// Mitsubishi GX Works2 project: 0708   PLC: Q02/Q02H

PROGRAM MAIN
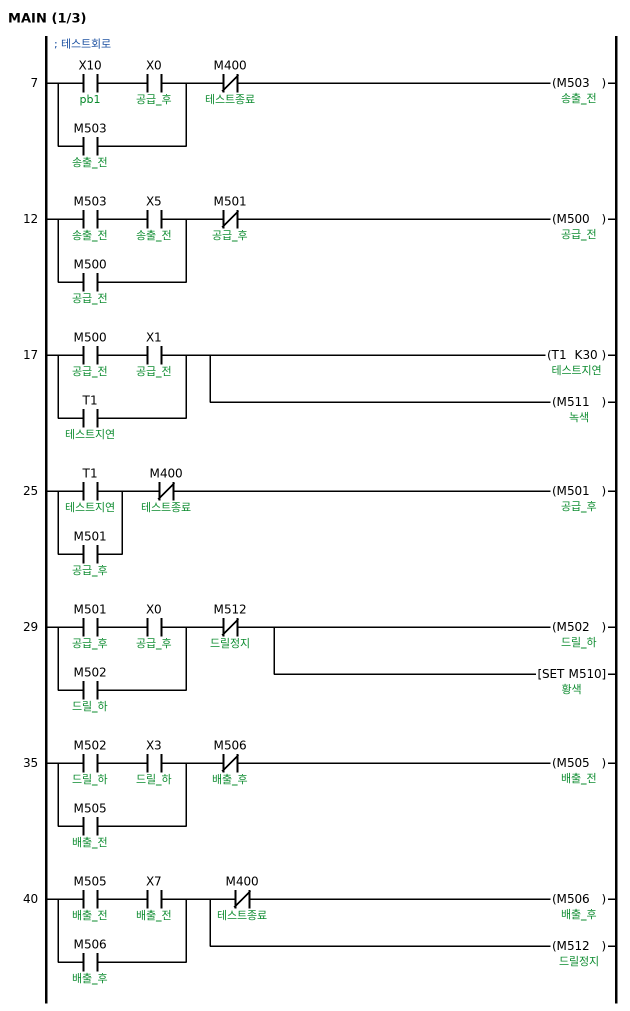
; 테스트회로
7     LD      X10  ; pb1
      AND     X0  ; 공급_후
      OR      M503  ; 송출_전
      ANI     M400  ; 테스트종료
      OUT     M503  ; 송출_전
12    LD      M503  ; 송출_전
      AND     X5  ; 송출_전
      OR      M500  ; 공급_전
      ANI     M501  ; 공급_후
      OUT     M500  ; 공급_전
17    LD      M500  ; 공급_전
      AND     X1  ; 공급_전
      OR      T1  ; 테스트지연
      OUT     T1 K30  ; 테스트지연
      OUT     M511  ; 녹색
25    LD      T1  ; 테스트지연
      OR      M501  ; 공급_후
      ANI     M400  ; 테스트종료
      OUT     M501  ; 공급_후
29    LD      M501  ; 공급_후
      AND     X0  ; 공급_후
      OR      M502  ; 드릴_하
      ANI     M512  ; 드릴정지
      OUT     M502  ; 드릴_하
      SET     M510  ; 황색
35    LD      M502  ; 드릴_하
      AND     X3  ; 드릴_하
      OR      M505  ; 배출_전
      ANI     M506  ; 배출_후
      OUT     M505  ; 배출_전
40    LD      M505  ; 배출_전
      AND     X7  ; 배출_전
      OR      M506  ; 배출_후
      MPS
      ANI     M400  ; 테스트종료
      OUT     M506  ; 배출_후
      MPP
      OUT     M512  ; 드릴정지
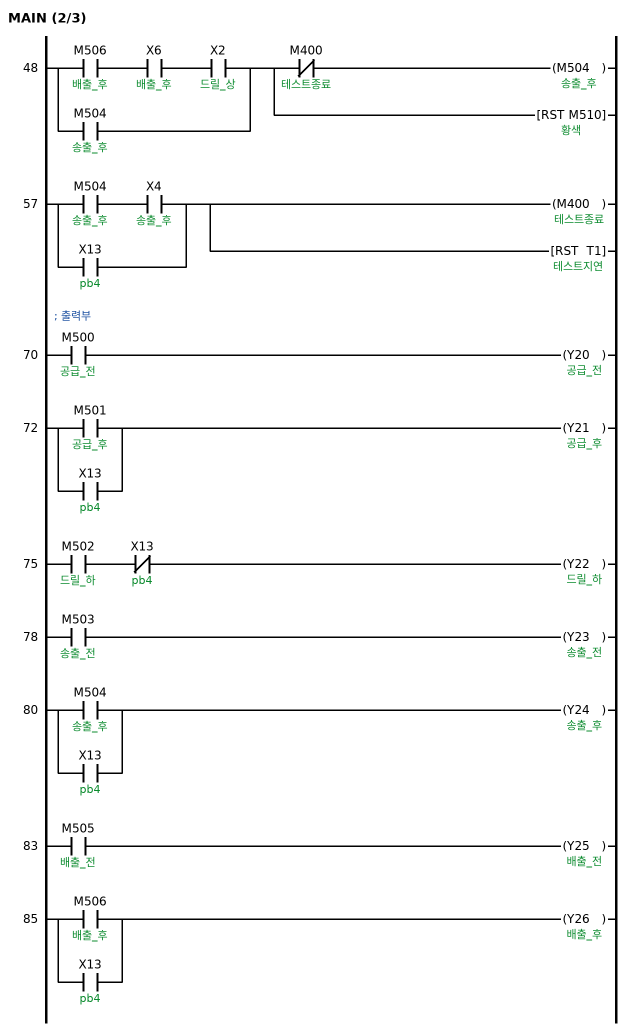
48    LD      M506  ; 배출_후
      AND     X6  ; 배출_후
      AND     X2  ; 드릴_상
      OR      M504  ; 송출_후
      MPS
      ANI     M400  ; 테스트종료
      OUT     M504  ; 송출_후
      MPP
      RST     M510  ; 황색
57    LD      M504  ; 송출_후
      AND     X4  ; 송출_후
      OR      X13  ; pb4
      OUT     M400  ; 테스트종료
      RST     T1  ; 테스트지연
; 출력부
70    LD      M500  ; 공급_전
      OUT     Y20  ; 공급_전
72    LD      M501  ; 공급_후
      OR      X13  ; pb4
      OUT     Y21  ; 공급_후
75    LD      M502  ; 드릴_하
      ANI     X13  ; pb4
      OUT     Y22  ; 드릴_하
78    LD      M503  ; 송출_전
      OUT     Y23  ; 송출_전
80    LD      M504  ; 송출_후
      OR      X13  ; pb4
      OUT     Y24  ; 송출_후
83    LD      M505  ; 배출_전
      OUT     Y25  ; 배출_전
85    LD      M506  ; 배출_후
      OR      X13  ; pb4
      OUT     Y26  ; 배출_후
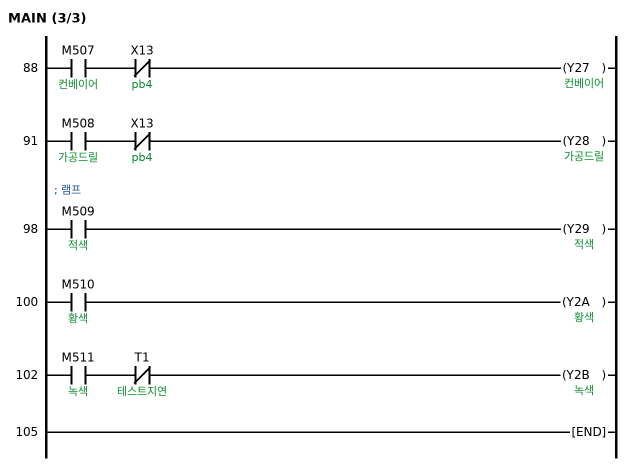
88    LD      M507  ; 컨베이어
      ANI     X13  ; pb4
      OUT     Y27  ; 컨베이어
91    LD      M508  ; 가공드릴
      ANI     X13  ; pb4
      OUT     Y28  ; 가공드릴
; 램프
98    LD      M509  ; 적색
      OUT     Y29  ; 적색
100   LD      M510  ; 황색
      OUT     Y2A  ; 황색
102   LD      M511  ; 녹색
      ANI     T1  ; 테스트지연
      OUT     Y2B  ; 녹색
105   END
END_PROGRAM

PROGRAM MAIN1
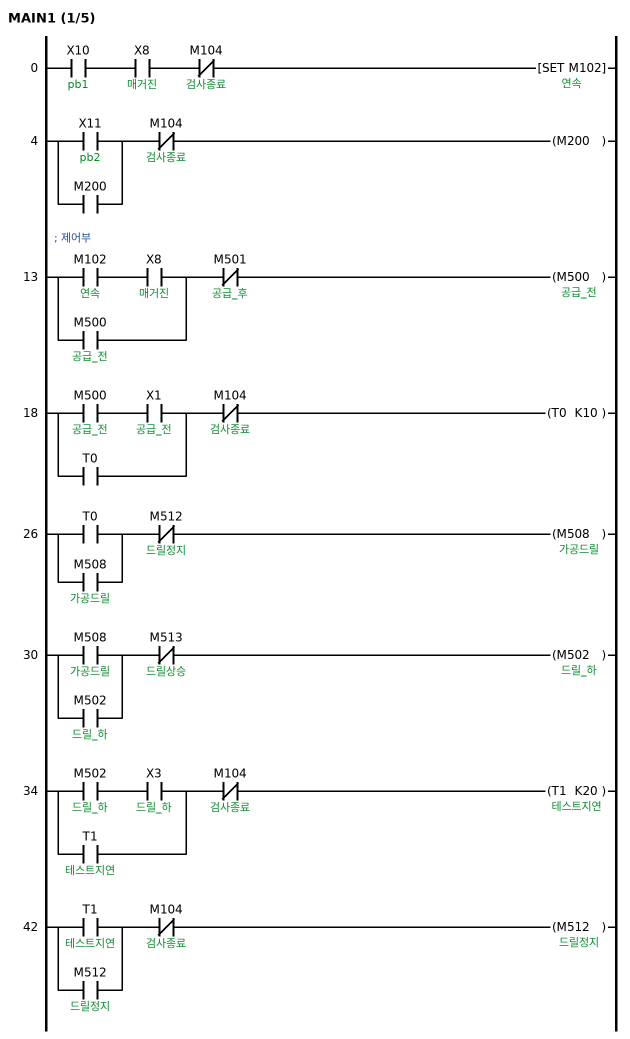
0     LD      X10  ; pb1
      AND     X8  ; 매거진
      ANI     M104  ; 검사종료
      SET     M102  ; 연속
4     LD      X11  ; pb2
      OR      M200
      ANI     M104  ; 검사종료
      OUT     M200
; 제어부
13    LD      M102  ; 연속
      AND     X8  ; 매거진
      OR      M500  ; 공급_전
      ANI     M501  ; 공급_후
      OUT     M500  ; 공급_전
18    LD      M500  ; 공급_전
      AND     X1  ; 공급_전
      OR      T0
      ANI     M104  ; 검사종료
      OUT     T0 K10
26    LD      T0
      OR      M508  ; 가공드릴
      ANI     M512  ; 드릴정지
      OUT     M508  ; 가공드릴
30    LD      M508  ; 가공드릴
      OR      M502  ; 드릴_하
      ANI     M513  ; 드릴상승
      OUT     M502  ; 드릴_하
34    LD      M502  ; 드릴_하
      AND     X3  ; 드릴_하
      OR      T1  ; 테스트지연
      ANI     M104  ; 검사종료
      OUT     T1 K20  ; 테스트지연
42    LD      T1  ; 테스트지연
      OR      M512  ; 드릴정지
      ANI     M104  ; 검사종료
      OUT     M512  ; 드릴정지
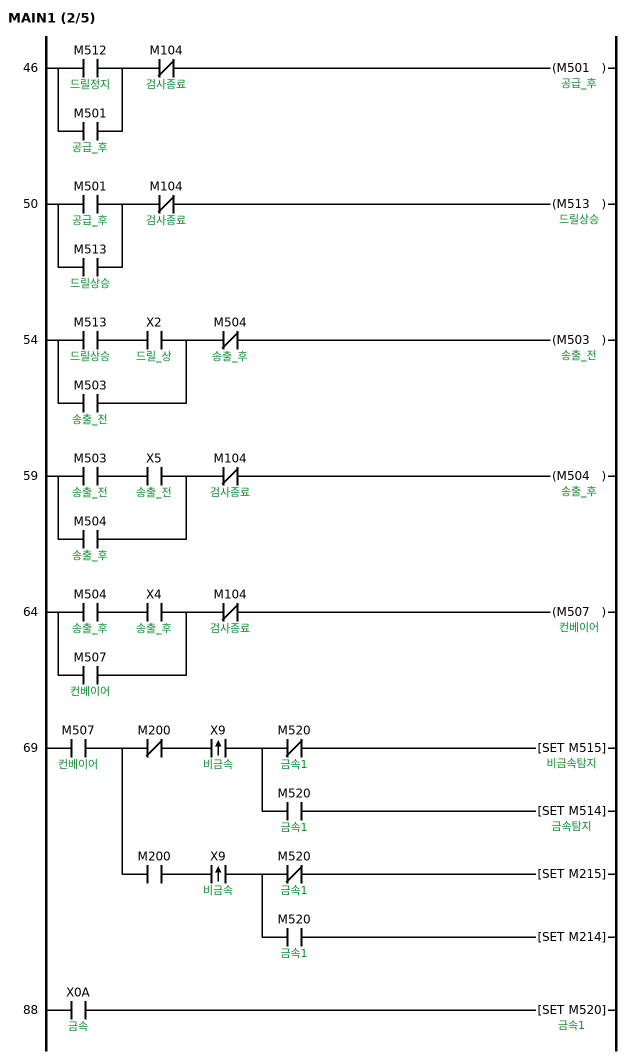
46    LD      M512  ; 드릴정지
      OR      M501  ; 공급_후
      ANI     M104  ; 검사종료
      OUT     M501  ; 공급_후
50    LD      M501  ; 공급_후
      OR      M513  ; 드릴상승
      ANI     M104  ; 검사종료
      OUT     M513  ; 드릴상승
54    LD      M513  ; 드릴상승
      AND     X2  ; 드릴_상
      OR      M503  ; 송출_전
      ANI     M504  ; 송출_후
      OUT     M503  ; 송출_전
59    LD      M503  ; 송출_전
      AND     X5  ; 송출_전
      OR      M504  ; 송출_후
      ANI     M104  ; 검사종료
      OUT     M504  ; 송출_후
64    LD      M504  ; 송출_후
      AND     X4  ; 송출_후
      OR      M507  ; 컨베이어
      ANI     M104  ; 검사종료
      OUT     M507  ; 컨베이어
69    LD      M507  ; 컨베이어
      MPS
      ANI     M200
      ANDP    X9  ; 비금속
      MPS
      ANI     M520  ; 금속1
      SET     M515  ; 비금속탐지
      MPP
      AND     M520  ; 금속1
      SET     M514  ; 금속탐지
      MPP
      AND     M200
      ANDP    X9  ; 비금속
      MPS
      ANI     M520  ; 금속1
      SET     M215
      MPP
      AND     M520  ; 금속1
      SET     M214
88    LD      X0A  ; 금속
      SET     M520  ; 금속1
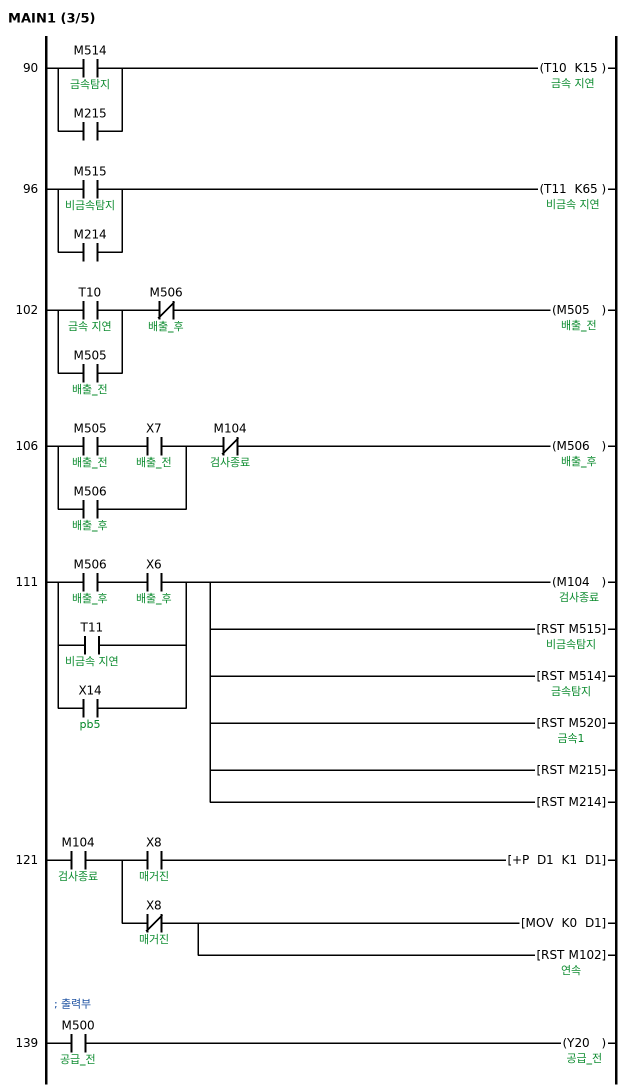
90    LD      M514  ; 금속탐지
      OR      M215
      OUT     T10 K15  ; 금속 지연
96    LD      M515  ; 비금속탐지
      OR      M214
      OUT     T11 K65  ; 비금속 지연
102   LD      T10  ; 금속 지연
      OR      M505  ; 배출_전
      ANI     M506  ; 배출_후
      OUT     M505  ; 배출_전
106   LD      M505  ; 배출_전
      AND     X7  ; 배출_전
      OR      M506  ; 배출_후
      ANI     M104  ; 검사종료
      OUT     M506  ; 배출_후
111   LD      M506  ; 배출_후
      AND     X6  ; 배출_후
      OR      T11  ; 비금속 지연
      OR      X14  ; pb5
      OUT     M104  ; 검사종료
      RST     M515  ; 비금속탐지
      RST     M514  ; 금속탐지
      RST     M520  ; 금속1
      RST     M215
      RST     M214
121   LD      M104  ; 검사종료
      MPS
      AND     X8  ; 매거진
      +P      D1 K1 D1
      MPP
      ANI     X8  ; 매거진
      MOV     K0 D1
      RST     M102  ; 연속
; 출력부
139   LD      M500  ; 공급_전
      OUT     Y20  ; 공급_전
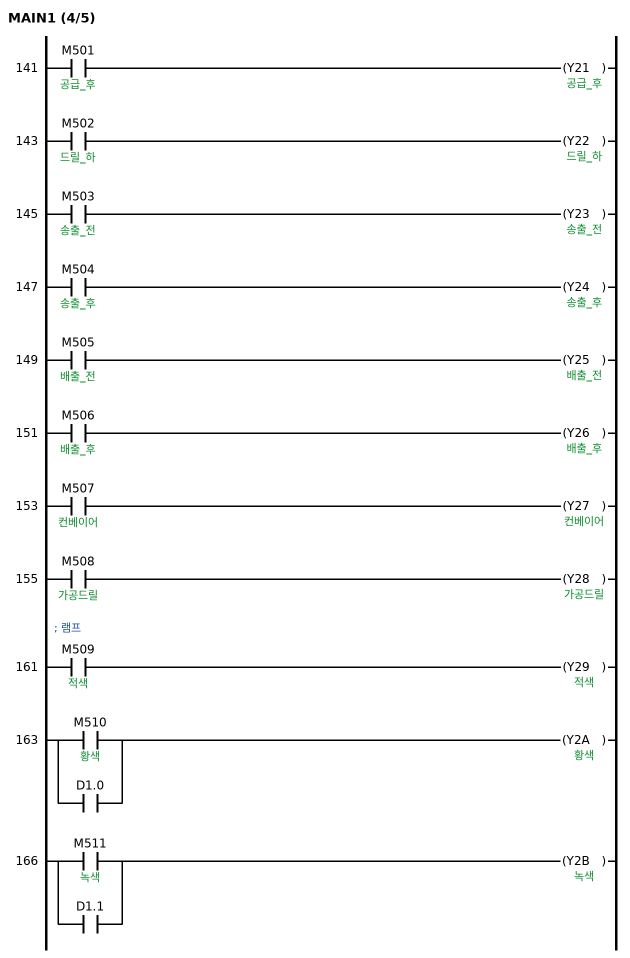
141   LD      M501  ; 공급_후
      OUT     Y21  ; 공급_후
143   LD      M502  ; 드릴_하
      OUT     Y22  ; 드릴_하
145   LD      M503  ; 송출_전
      OUT     Y23  ; 송출_전
147   LD      M504  ; 송출_후
      OUT     Y24  ; 송출_후
149   LD      M505  ; 배출_전
      OUT     Y25  ; 배출_전
151   LD      M506  ; 배출_후
      OUT     Y26  ; 배출_후
153   LD      M507  ; 컨베이어
      OUT     Y27  ; 컨베이어
155   LD      M508  ; 가공드릴
      OUT     Y28  ; 가공드릴
; 램프
161   LD      M509  ; 적색
      OUT     Y29  ; 적색
163   LD      M510  ; 황색
      OR      D1.0
      OUT     Y2A  ; 황색
166   LD      M511  ; 녹색
      OR      D1.1
      OUT     Y2B  ; 녹색
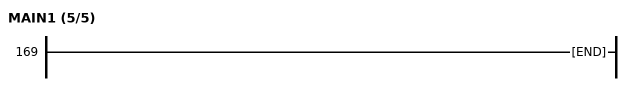
169   END
END_PROGRAM

// device comments not shown above
X12  ; pb3
M100  ; 테스트
M101  ; 단속
M103  ; 초기화
M401  ; 금속종료
M402  ; 비금속종료
M600  ; blink
M601  ; blink_0.5
M700  ; 공급_전2
M701  ; 공급_후2
M702  ; 드릴_하2
M703  ; 송출_전2
M704  ; 송출_후2
M705  ; 배출_전2
M706  ; 배출_후2
M707  ; 컨베이어
M708  ; 가공드릴2
M709  ; 적색2
M710  ; 황색2
M711  ; 녹색2
